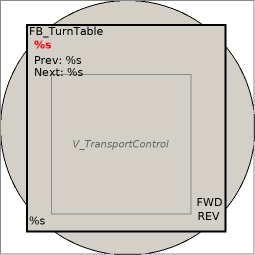
VISUALIZATION V_TurnTable  // 255x255
VAR_IN_OUT
	{attribute 'VAR_IN_OUT_AS_POINTER'}
	fbFunction		: FB_TurnTable;	
END_VAR
    Ellipse (0,0 255x255), colour toggle: fbFunction.FunctionInterface.Out.FunctionOrders.ReqDriveRun OR fbFunction.FunctionInterface.Out.FunctionOrders.ReqDriveRun_34
    Rectangle (26,24 200x208), colour toggle: fbFunction.HW_Outputs.Drive_Run_CW OR fbFunction.HW_Outputs.Drive_Run_CCW
    Rectangle (26,211 200x20), "%s", text variable: fbFunction.ConfigFunction.FunctionName
    Label (26,24 200x15), "FB_TurnTable"
    Label (192,196 35x13), "FWD", invisible if: NOT fbFunction.HW_Outputs.Drive_Run_CW
    Label (191,209 35x15), "REV", invisible if: NOT fbFunction.HW_Outputs.Drive_Run_CCW
    Frame (51,74 140x140)
        shows V_TransportControl(TransportControl := fbFunction.fbTransportControl, ZoneData := fbFunction.ZoneData[1])
    Rectangle (31,37 194x16), "%s", tooltip "%s", text variable: fbFunction.FunctionData.ErrorData.Error.ErrorCode.Conv, invisible if: fbFunction.FunctionData.ErrorData.ErrorState = E_ErrorState.OPERATIONAL
        p4168582468: fbFunction.FunctionData.ErrorData.Error.ErrorParam
    Rectangle (31,54 200x13), "Prev: %s", tooltip "FunctionInterface.in.ePrevFunctionNumber", text variable: fbFunction.FunctionInterface.In.ePrevFunctionNumber
    Rectangle (31,66 200x13), "Next: %s", tooltip "FunctionInterface.in.eNextFunctionNumber", text variable: fbFunction.FunctionInterface.In.eNextFunctionNumber
END_VISUALIZATION

(* stored: Version 1.1.0.1, ProductVersion 3.1.4024.9
   Visu V_TurnTable: Id {bdee249d-c6b2-40b3-9d03-42d5a7256562} *)
